// TIA Portal project "openness_project_20230911_201755" (V17)

(* hardware
DEVICE "n0001-zp001-el001-k30001"  S7-1500 station
   slot 0: "Rail_0"  Rack  6ES7 590-1***0-0AA0
   slot 1: "n0001-zp001-el001-k30001"  CPU 1517F-3 PN/DP  6ES7 517-3FP00-0AB0  V2.9
      slot 3: "CPU display_1"  6ES7591-1BA00-0AA0
      slot 32768: "PROFINET interface_1"  X1
         slot 32769: "Port_1"  X1 P1
         slot 32770: "Port_2"  X1 P2
      slot 33024: "PROFINET interface_2"  X2
         slot 33025: "Port_1"  X2 P1
      slot 33280: "DP interface_1"  X3
      slot 34817: "Virtual CP interface port_1"  Virtual CP interface port  Virtual CP interface port
   slot 2: "n0001-zp001-el001-k30002"  CM 1542-1  6GK7 542-1AX00-0XE0  V3.0
DEVICE "n0005-lv008-el001-k30001"  ET 200SP-Station
   slot 0: "Rack_0"  Rack  6ES5 710-8MAx1
   slot 0: "n0005-lv008-el001-k30001"  IM 155-6 PN ST  6ES7 155-6AU01-0BN0  V4.2
   slot 1: "-K30002"  DI 16x24VDC ST  6ES7 131-6BH01-0BA0  V0.0
      slot 1: "-K30002"  DI 16x24VDC ST
   slot 2: "-K30003"  F-DI 8x24VDC HF  6ES7 136-6BA00-0CA0  V1.0
      slot 1: "-K30003"  F-DI 8x24VDC HF
   slot 3: "-K30004"  F-DI 8x24VDC HF  6ES7 136-6BA00-0CA0  V1.0
      slot 1: "-K30004"  F-DI 8x24VDC HF
   slot 4: "-K30005"  F-DQ 4x24VDC/2A PM HF  6ES7 136-6DB00-0CA0  V2.0
      slot 1: "-K30005"  F-DQ 4x24VDC/2A PM HF
   slot 5: "-K30006"  F-DQ 4x24VDC/2A PM HF  6ES7 136-6DB00-0CA0  V2.0
      slot 1: "-K30006"  F-DQ 4x24VDC/2A PM HF
   slot 6: "Server module_1"  Server module  6ES7 193-6PA00-0AA0  V1.1
      slot 1: "Server module_1"  Server module
   slot 127: "BA 2xRJ45"  BA 2xRJ45  6ES7 193-6AR00-0AA0  V0.0
      slot 1: "Port_1"  X1 P1 R  6ES7 193-6AR00-0AA0  V0.0
      slot 2: "Port_2"  X1 P2 R  6ES7 193-6AR00-0AA0  V0.0
DEVICE "n0013-uf317-xn10"  GSD.Device.PN
   slot 0: "Rack"  Rack  V1.0
   slot 0: "n0013-uf317-xn10"  55556 MVK-MPNIO F DI16/8  55556
      slot 0: "55556 MVK-MPNIO F DI16/8_1"  55556 MVK-MPNIO F DI16/8
      slot 1: "Power module_1"  Power module
         slot 0: "Power module"  Power module
      slot 1: "55556 MVK-MPNIO F DI16/8"  55556 MVK-MPNIO F DI16/8
         slot 1: "Port 1"  Port 1
         slot 2: "Port 2"  Port 2
   slot 2: "-XN10"  FS Data
      slot 0: "-XN10"  FS Data
*)

// ===== PLC "n0001-zp001-el001-k30001"  CPU 1517F-3 PN/DP =====

DATA_BLOCK "Main_Safety_RTG1_DB"   // DB1, F_DB
{ S7_Optimized_Access := 'TRUE' }
NAME : FUSI
VERSION : 0.1
// stored: InstanceOfName Main_Safety_RTG1
"Main_Safety_RTG1"
BEGIN
END_DATA_BLOCK

FUNCTION_BLOCK "Main_Safety_RTG1"   // FB1, F_FBD
{ S7_Optimized_Access := 'TRUE' }
BEGIN
END_FUNCTION_BLOCK

ORGANIZATION_BLOCK "Main"   // OB1, LAD, ProgramCycle
TITLE = "Main Program Sweep (Cycle)"
{ S7_Optimized_Access := 'TRUE' }
VERSION : 0.1
   VAR_INPUT
      Initial_Call : Bool;   // Initial call of this OB
      Remanence : Bool;   // =True, if remanent data are available
   END_VAR
BEGIN
END_ORGANIZATION_BLOCK